FUNCTION_BLOCK FB 251
TITLE =G151M FRESH AIR LOUVER GERM 3
//COPYRIGHT:    (C) 2009  BUHLER AG, CH-9240 UZWIL, SWITZERLAND
//
//PRODUCT:      WinCoS_BIW01_09
//
//TITLE:        FRESH AIR LOUVER GERM 3
//                Machine group control
//                Maschinengruppensteuerung
//
//--------------------------------------------------------------------------------
//
//IDENT:        AUTHOR:             DEPT:                              DATE:
//
//P01_FB251.1.0 K.Renz              CSB41                              13.Jan.2010
//             1st Release
//
//--------------------------------------------------------------------------------
//
//PURPOSE:
//
//MANUAL :
//
//RESTRICTIONS:
//
//--------------------------------------------------------------------------------
AUTHOR : KR
FAMILY : USW
VERSION : 9.9


VAR
  Gr : FB 10;	//Standard interface to group
  InOutValue1 : DINT ;	//Data for user
  InOutValue2 : DINT ;	//Data for user
  OutWayConflict : BOOL ;	//Data for user
  OutSelectionOk : BOOL ;	//Data for user
  CmdNewValue : BOOL ;	//Data for user
  CmdNewJob : BOOL ;	//Data for user
  OutCodeOK : BOOL ;	//Data for user
  InEndOfJob : BOOL ;	//Data for user
  staWayOk : BOOL ;	//Data for user
  EdgeStartRelease : BOOL ;	//Data for user
  USW8 : BOOL ;	//Data for user
  USW9 : BOOL ;	//Data for user
  USW10 : BOOL ;	//Data for user
  USW11 : BOOL ;	//Data for user
  USW12 : BOOL ;	//Data for user
  USW13 : BOOL ;	//Data for user
  USW14 : BOOL ;	//Data for user
  USW15 : BOOL ;	//Data for user
  A_2351_BZS01 : FB 14;	// DigInpCont
  A_2351_BZS02 : FB 14;	// DigInpCont
  A_2351_MXZ01 : FB 20;	// VLS4Ctrl
  A_2352_BZS01 : FB 14;	// DigInpCont
  A_2352_BZS02 : FB 14;	// DigInpCont
  A_2352_MXZ01 : FB 20;	// VLS4Ctrl
END_VAR
VAR_TEMP
  tmpEnable : BOOL ;
  tmpFlag : BOOL ;
  tmpCmdNext : BOOL ;
  tmpLocal : BOOL ;
  tmpAspOk : BOOL ;
  tmpHWStop : BOOL ;
  tmpInstanzDBNo : INT ;
END_VAR
BEGIN
NETWORK
TITLE =



NETWORK
TITLE =Read command from group control
//Parameter
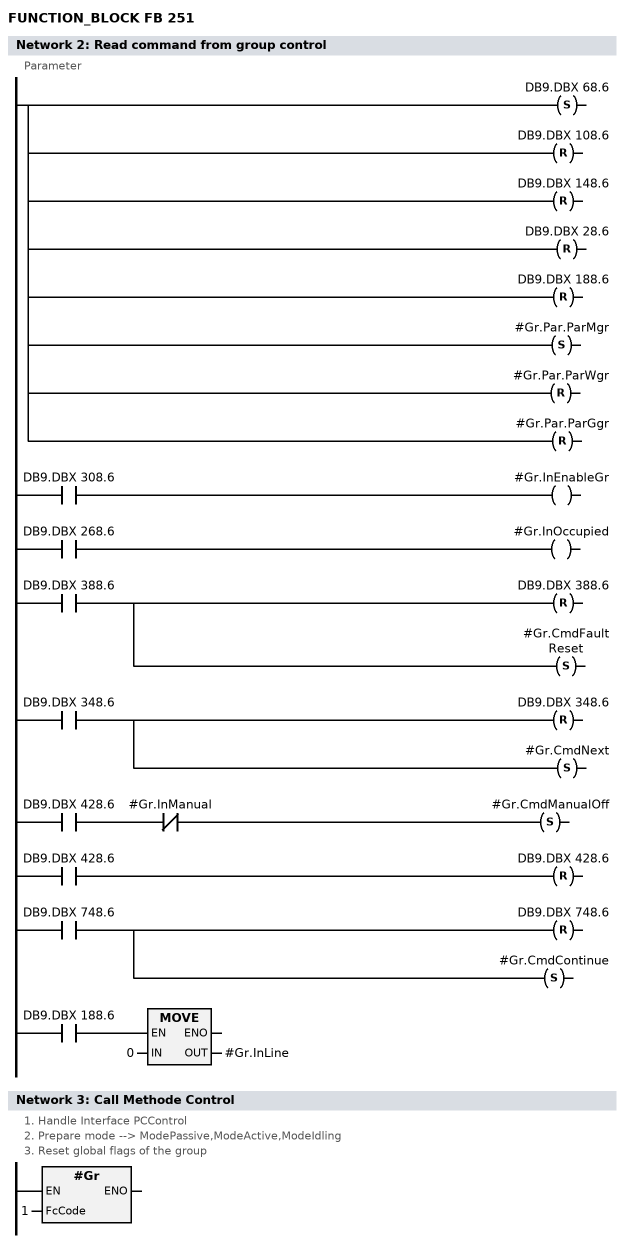
      SET   ;
      S     DB9.DBX   68.6;
      R     DB9.DBX  108.6;
      R     DB9.DBX  148.6;
      R     DB9.DBX   28.6;
      R     DB9.DBX  188.6;
      S     #Gr.Par.ParMgr;
      R     #Gr.Par.ParWgr;
      R     #Gr.Par.ParGgr;
//Command
      A     DB9.DBX  308.6;
      =     #Gr.InEnableGr;
      A     DB9.DBX  268.6;
      =     #Gr.InOccupied;
      A     DB9.DBX  388.6;
      R     DB9.DBX  388.6;
      S     #Gr.CmdFaultReset;
      A     DB9.DBX  348.6;
      R     DB9.DBX  348.6;
      S     #Gr.CmdNext;

      A     DB9.DBX  428.6;
      AN    #Gr.InManual;
      S     #Gr.CmdManualOff;
      A     DB9.DBX  428.6;
      R     DB9.DBX  428.6;

//      U     "GCS7_GrCtrlDB".CmdManualOff[151]
//      O     "GCS7_GrCtrlDB".OutOccupied[151]
//      R     "GCS7_GrCtrlDB".CmdManualOff[151]
//      S     #Gr.CmdManualOff

      A     DB9.DBX  748.6;
      R     DB9.DBX  748.6;
      S     #Gr.CmdContinue;
//Init Line Number
      A     DB9.DBX  188.6;
      JCN   WE00;
      L     0;
      T     #Gr.InLine;
WE00: NOP   0;
NETWORK
TITLE =Call Methode Control
// 1. Handle Interface PCControl
// 2. Prepare mode --> ModePassive,ModeActive,ModeIdling
// 3. Reset global flags of the group
      CALL #Gr (
           FcCode                   := 1);
NETWORK
TITLE =Restart Idling Time

      L     #Gr.Par.ParIdling;
      L     2;
      >=I   ;
      JC    IdTm;
      T     #Gr.Par.ParIdling;
IdTm: NOP   0;
      CLR   ;
      S     #Gr.CmdRestartIdling;
NETWORK
TITLE =Prepare global flags



NETWORK
TITLE =Set Pattern (Target position)

      A     #Gr.InManual;
      JC    ILO6;
      L     0; // 0.0%
      O     DB819.DBX  111.6;
      O     DB819.DBX  111.0;
      JC    PE;
      A     DB909.DBX  410.0;
      O(    ;
      A     DB909.DBX  412.1; // germinating Process finished
      AN    DB819.DBX  111.4;
      )     ;
      JCN   M003;
      NOP   0;
//BRT100310      L     "MAL1S019Par".StepAct.PosFreshAirFlapBasic
//      L     "MAL1S019Par".Par.ParIntMachine.TargetPosFreshAir    //BRT100310
//      L     10                          // convert to 0.1%
//      *I
PE:   NOP   0;

      A     DB251.DBX  131.5;
      JC    Man1;
      L     DB909.DBW  352; //BRT100310
      L     10; // convert to 0.1%
      *I    ;
      T     #A_2351_MXZ01.InPositionMiddle; // setpoint element
//-> 26.02.2014 IS. Start regulating from current position when switch to automatic
Man1: L     #A_2351_MXZ01.InPositionMiddle;
      L     10;
      /D    ;
      T     DB909.DBW  352;
//<-
      NOP   0;

      A     DB251.DBX  259.5;
      JC    Man2;
      L     DB909.DBW  254; // Target Position FreshAir 2
      L     10; // convert to 0.1%
      *I    ;
      T     #A_2352_MXZ01.InPositionMiddle; // setpoint element
//-> 26.02.2014 IS. Start regulating from current position when switch to automatic
Man2: L     #A_2352_MXZ01.InPositionMiddle;
      L     10;
      /D    ;
      T     DB909.DBW  254;
//<-
M003: NOP   0;
      JU    En06;
ILO6: NOP   0;
      L     DB909.DBW  230;
      L     10; // convert to 0.1%
      *I    ;
      T     #A_2351_MXZ01.InPositionMiddle; // setpoint element
      T     #A_2352_MXZ01.InPositionMiddle; // setpoint element
En06: NOP   0;



NETWORK
TITLE =Interlocking WayOk



NETWORK
TITLE =Interlocking Autostart

      CLR   ;
      R     #Gr.OutAutostart;
NETWORK
TITLE =Interlocking Enable
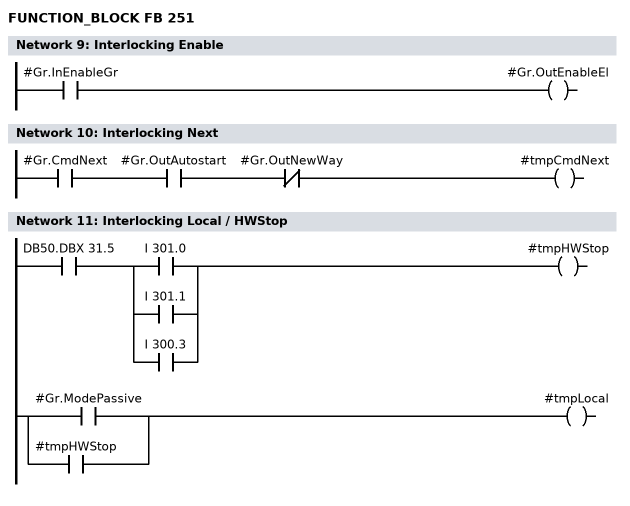

      A     #Gr.InEnableGr;
      =     #Gr.OutEnableEl;

NETWORK
TITLE =Interlocking Next

      A     #Gr.CmdNext;
      A     #Gr.OutAutostart;
      AN    #Gr.OutNewWay;
      =     #tmpCmdNext;

NETWORK
TITLE =Interlocking Local / HWStop

      A     DB50.DBX   31.5;
//BRT100310 - HW-Stop nur bei NOT-AUS +C23 oder Customer, nicht bei NOT-AUS Maschine!
      A(    ;
      O     I    301.0;
      O     I    301.1;
      O     I    300.3;
      )     ;
      =     #tmpHWStop;

      A     #Gr.ModePassive;
      O     #tmpHWStop;
      =     #tmpLocal;

NETWORK
TITLE ==A-2351-BZS01 : FRESH AIR FLAP 1 100% CIRCULATION AIR

      NOP   0;
//-InLocal---
      A     #tmpLocal;
      =     #A_2351_BZS01.InLocal;
//
//-Monitoring---
      CLR   ;
      =     #A_2351_BZS01.InMonTrue;
      CLR   ;
      =     #A_2351_BZS01.InMonFalse;
//
//-PreAlarm---
      CLR   ;
      =     #A_2351_BZS01.InPreAlarmTrue;
      CLR   ;
      =     #A_2351_BZS01.InPreAlarmFalse;
//
//-Additional commands---
//      CLR
//      S     #A_2351_BZS01.CmdRunTimeOutTime
//
//-Read inputs---
      A     I    364.6;
      =     #A_2351_BZS01.InpTrue;
      A     DB51.DBX    4.5;
      =     #A_2351_BZS01.InDPFault;
//
//-Set Parameters---
//
//-Call object control---
      CALL #A_2351_BZS01 ;
//
//-Write outputs---
NETWORK
TITLE ==A-2351-BZS02 : FRESH AIR FLAP 1 100% FRESH AIR

      NOP   0;
//-InLocal---
      A     #tmpLocal;
      =     #A_2351_BZS02.InLocal;
//
//-Monitoring---
      CLR   ;
      =     #A_2351_BZS02.InMonTrue;
      CLR   ;
      =     #A_2351_BZS02.InMonFalse;
//
//-PreAlarm---
      CLR   ;
      =     #A_2351_BZS02.InPreAlarmTrue;
      CLR   ;
      =     #A_2351_BZS02.InPreAlarmFalse;
//
//-Additional commands---
//      CLR
//      S     #A_2351_BZS02.CmdRunTimeOutTime
//
//-Read inputs---
      A     I    364.7;
      =     #A_2351_BZS02.InpTrue;
      A     DB51.DBX    4.5;
      =     #A_2351_BZS02.InDPFault;
//
//-Set Parameters---
//
//-Call object control---
      CALL #A_2351_BZS02 ;
//
//-Write outputs---
NETWORK
TITLE ==A-2351-MXZ01 : FRESH AIR FLAP 1

      NOP   0;
//-InLocal---
      A(    ;
      A     #tmpLocal;
      O     ;
      A     #Gr.InManual;
      AN    #Gr.InOutAutostartMan;
      )     ;
      A     #A_2351_MXZ01.StLN;
      =     #A_2351_MXZ01.InLocal;

//-Interlocking---
      A     #A_2351_MXZ01.Par.ParManual;
      A     #A_2351_MXZ01.InManual;
      JC    man1;
      A(    ;
      L     0;
      L     #A_2351_MXZ01.InPositionMiddle; // setpoint element
      ==I   ;
      )     ;
      A(    ;
      A     #Gr.InManual;
      A     #Gr.InOutAutostartMan;
      ON    #Gr.InManual;
      )     ;
      A     #Gr.OutEnableEl;
      =     #A_2351_MXZ01.InLN;

      A(    ;
      L     #A_2351_MXZ01.InPositionMiddle; // setpoint element
      L     0;
      >I    ;
      )     ;
      A(    ;
      L     #A_2351_MXZ01.InPositionMiddle; // setpoint element
      L     1000; // 100,0%
      <I    ;
      )     ;
      A(    ;
      A     #Gr.InManual;
      A     #Gr.InOutAutostartMan;
      ON    #Gr.InManual;
      )     ;
      A     #Gr.OutEnableEl;
      S     #A_2351_MXZ01.CmdMiddle1;

      CLR   ;
      =     #A_2351_MXZ01.CmdMiddle2;

      A(    ;
      AN    #Gr.InOccupied;
      AN    #Gr.InManual;
      )     ;
      O(    ;
      L     #A_2351_MXZ01.InPositionMiddle; // setpoint element
      L     1000; // 100,0%
      >=I   ;
      )     ;
      A(    ;
      A     #Gr.InManual;
      A     #Gr.InOutAutostartMan;
      ON    #Gr.InManual;
      )     ;
      A     #Gr.OutEnableEl;
      S     #A_2351_MXZ01.CmdHN;
man1: NOP   0;
//
//-Read inputs---
//====>BRT060310 - Regeln auf Zeit, ohne Auswertung Rückmeldung
      A     I    364.6;
      =     DB251.DBX  130.4;
      CLR   ;
      =     DB251.DBX  130.5;
      A     I    364.7;
      =     DB251.DBX  130.7;

//      U     #A_2351_BZS02.StTrue        // 100% Frischluft
//      SPBN  FL1
//      L     1000
//      SPA   INP1
//FL1:  NOP   0
//      U     #A_2351_BZS01.StTrue        // 100% Umluft
//      SPBN  RL1
//      L     0
//      SPA   INP1
//RL1:  NOP   0
//      L     "A_2351_BEE01_AI1"
//INP1: T     #A_2351_MXZ01.InpPosition
//<====BRT060310
//BRT110310      U     "PLC_SystemDB".HardwareStop.Germinating_3
      A     #tmpHWStop; //BRT110310
      =     #A_2351_MXZ01.InHWStop;
      A     DB51.DBX    4.5;
      =     #A_2351_MXZ01.InDPFault;
//
//-Set Parameters---
//
//-Call object control---
      CALL #A_2351_MXZ01 ;
//
//-Write outputs---
      A     #A_2351_MXZ01.OutpLN;
      =     Q    364.5;
      A     #A_2351_MXZ01.OutpHN;
      =     Q    364.4;

NETWORK
TITLE ==A-2352-BZS02 : FRESH AIR FLAP 2 100% FRESH AIR

      NOP   0;
//-InLocal---
      A     #tmpLocal;
      =     #A_2352_BZS02.InLocal;
//
//-Monitoring---
      CLR   ;
      =     #A_2352_BZS02.InMonTrue;
      CLR   ;
      =     #A_2352_BZS02.InMonFalse;
//
//-PreAlarm---
      CLR   ;
      =     #A_2352_BZS02.InPreAlarmTrue;
      CLR   ;
      =     #A_2352_BZS02.InPreAlarmFalse;
//
//-Additional commands---
//      CLR
//      S     #A_2352_BZS02.CmdRunTimeOutTime
//
//-Read inputs---
      A     I    365.3;
      =     #A_2352_BZS02.InpTrue;
      A     DB51.DBX    4.5;
      =     #A_2352_BZS02.InDPFault;
//
//-Set Parameters---
//
//-Call object control---
      CALL #A_2352_BZS02 ;
//
//-Write outputs---
NETWORK
TITLE ==A-2352-BZS01 : FRESH AIR FLAP 2 100% CIRCULATION AIR

      NOP   0;
//-InLocal---
      A     #tmpLocal;
      =     #A_2352_BZS01.InLocal;
//
//-Monitoring---
      CLR   ;
      =     #A_2352_BZS01.InMonTrue;
      CLR   ;
      =     #A_2352_BZS01.InMonFalse;
//
//-PreAlarm---
      CLR   ;
      =     #A_2352_BZS01.InPreAlarmTrue;
      CLR   ;
      =     #A_2352_BZS01.InPreAlarmFalse;
//
//-Additional commands---
//      CLR
//      S     #A_2352_BZS01.CmdRunTimeOutTime
//
//-Read inputs---
      A     I    365.2;
      =     #A_2352_BZS01.InpTrue;
      A     DB51.DBX    4.5;
      =     #A_2352_BZS01.InDPFault;
//
//-Set Parameters---
//
//-Call object control---
      CALL #A_2352_BZS01 ;
//
//-Write outputs---
NETWORK
TITLE ==A-2352-MXZ01 : FRESH AIR FLAP 2

      NOP   0;
//-InLocal---
      A(    ;
      A     #tmpLocal;
      O     ;
      A     #Gr.InManual;
      AN    #Gr.InOutAutostartMan;
      )     ;
      A     #A_2352_MXZ01.StLN;
      =     #A_2352_MXZ01.InLocal;

//-Interlocking---
      A     #A_2352_MXZ01.Par.ParManual;
      A     #A_2352_MXZ01.InManual;
      JC    man2;
      A(    ;
      L     0;
      L     #A_2352_MXZ01.InPositionMiddle; // setpoint element
      ==I   ;
      )     ;
      A(    ;
      A     #Gr.InManual;
      A     #Gr.InOutAutostartMan;
      ON    #Gr.InManual;
      )     ;
      A     #Gr.OutEnableEl;
      =     #A_2352_MXZ01.InLN;

      A(    ;
      L     #A_2352_MXZ01.InPositionMiddle; // setpoint element
      L     0;
      >I    ;
      )     ;
      A(    ;
      L     #A_2352_MXZ01.InPositionMiddle; // setpoint element
      L     1000; // 100,0%
      <I    ;
      )     ;
      A(    ;
      A     #Gr.InManual;
      A     #Gr.InOutAutostartMan;
      ON    #Gr.InManual;
      )     ;
      A     #Gr.OutEnableEl;
      S     #A_2352_MXZ01.CmdMiddle1;

      CLR   ;
      =     #A_2352_MXZ01.CmdMiddle2;

      A(    ;
      AN    #Gr.InOccupied;
      AN    #Gr.InManual;
      )     ;
      O(    ;
      L     #A_2352_MXZ01.InPositionMiddle; // setpoint element
      L     1000; // 100,0%
      >=I   ;
      )     ;
      A(    ;
      A     #Gr.InManual;
      A     #Gr.InOutAutostartMan;
      ON    #Gr.InManual;
      )     ;
      A     #Gr.OutEnableEl;
      S     #A_2352_MXZ01.CmdHN;
man2: NOP   0;
//
//-Read inputs---
//====>BRT060310 - Regeln auf Zeit, ohne Auswertung Rückmeldung
      A     I    365.2;
      =     DB251.DBX  258.4;
      CLR   ;
      =     DB251.DBX  258.5;
      A     I    365.3;
      =     DB251.DBX  258.7;

//      U     #A_2352_BZS02.StTrue        // 100% Frischluft
//      SPBN  FL2
//      L     1000
//      SPA   INP2
//FL2:  NOP   0
//      U     #A_2352_BZS01.StTrue        // 100% Umluft
//      SPBN  RL2
//      L     0
//      SPA   INP2
//RL2:  NOP   0
//      L     "A_2352_BEE01_AI1"
//INP2: T     #A_2352_MXZ01.InpPosition
//<====BRT100310
//BRT110310      U     "PLC_SystemDB".HardwareStop.Germinating_3
      A     #tmpHWStop; //BRT110310
      =     #A_2352_MXZ01.InHWStop;
      A     DB51.DBX    4.5;
      =     #A_2352_MXZ01.InDPFault;
//
//-Set Parameters---
//
//-Call object control---
      CALL #A_2352_MXZ01 ;
//
//-Write outputs---
      A     #A_2352_MXZ01.OutpLN;
      =     Q    365.1;
      A     #A_2352_MXZ01.OutpHN;
      =     Q    365.0;

NETWORK
TITLE =Test Fault
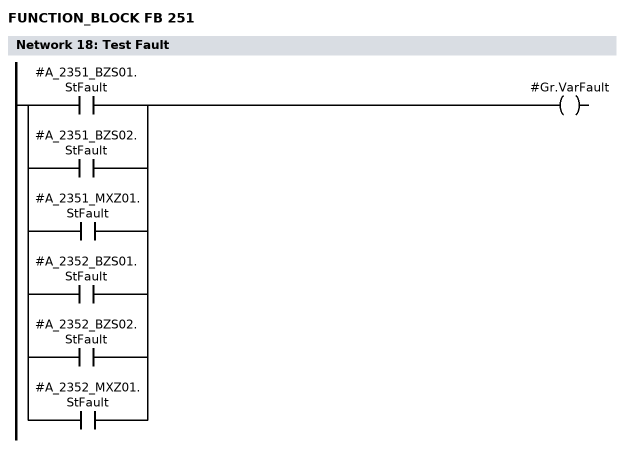

      A     #A_2351_BZS01.StFault;
      O     #A_2351_BZS02.StFault;
      O     #A_2351_MXZ01.StFault;
      O     #A_2352_BZS01.StFault;
      O     #A_2352_BZS02.StFault;
      O     #A_2352_MXZ01.StFault;
      =     #Gr.VarFault;
NETWORK
TITLE =Test Warning

      CLR   ;
      =     #Gr.OutWarning;
NETWORK
TITLE =Test Stopped
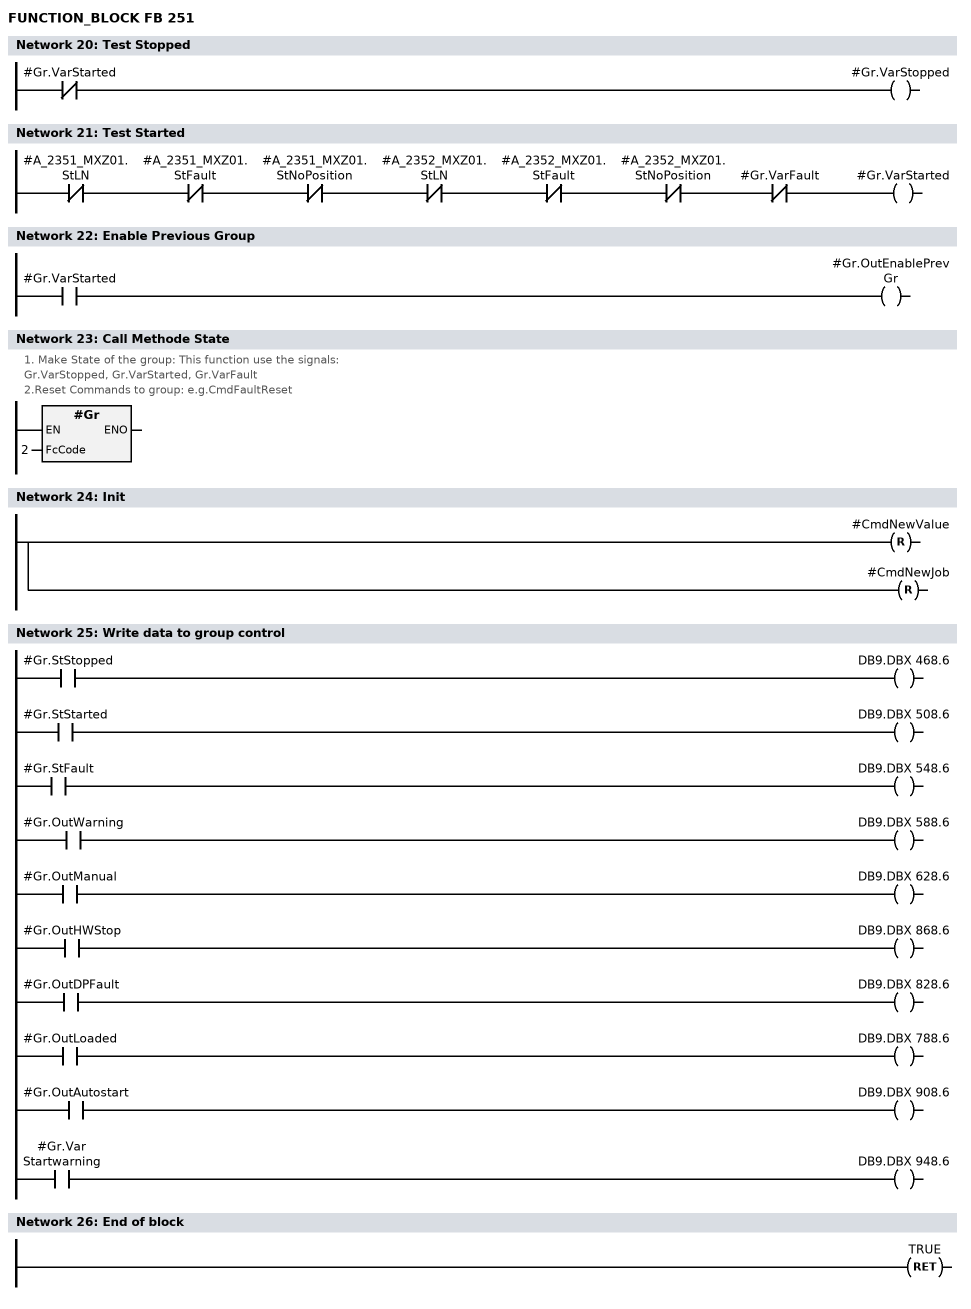

//BRT100310       U     #A_2351_MXZ01.StLN
//BRT100310       U     #A_2352_MXZ01.StLN
//BRT100310       UN    #Gr.VarFault
      AN    #Gr.VarStarted;
      =     #Gr.VarStopped;
NETWORK
TITLE =Test Started

      AN    #A_2351_MXZ01.StLN;
      AN    #A_2351_MXZ01.StFault;
      AN    #A_2351_MXZ01.StNoPosition;
      AN    #A_2352_MXZ01.StLN;
      AN    #A_2352_MXZ01.StFault;
      AN    #A_2352_MXZ01.StNoPosition;
//BRT100310      UN    #Gr.VarStopped
      AN    #Gr.VarFault;
      =     #Gr.VarStarted;
NETWORK
TITLE =Enable Previous Group

      A     #Gr.VarStarted;
      =     #Gr.OutEnablePrevGr;
NETWORK
TITLE =Call Methode State
//1. Make State of the group: This function use the signals:
//        Gr.VarStopped, Gr.VarStarted, Gr.VarFault
//2.Reset Commands to group: e.g.CmdFaultReset
      CALL #Gr (
           FcCode                   := 2);
NETWORK
TITLE =Init

      SET   ;
      R     #CmdNewValue;
      R     #CmdNewJob;
NETWORK
TITLE =Write data to group control

      A     #Gr.StStopped;
      =     DB9.DBX  468.6;
      A     #Gr.StStarted;
      =     DB9.DBX  508.6;
      A     #Gr.StFault;
      =     DB9.DBX  548.6;
      A     #Gr.OutWarning;
      =     DB9.DBX  588.6;
      A     #Gr.OutManual;
      =     DB9.DBX  628.6;
      A     #Gr.OutHWStop;
      =     DB9.DBX  868.6;
      A     #Gr.OutDPFault;
      =     DB9.DBX  828.6;
      A     #Gr.OutLoaded;
      =     DB9.DBX  788.6;
      A     #Gr.OutAutostart;
      =     DB9.DBX  908.6;
      A     #Gr.VarStartwarning;
      =     DB9.DBX  948.6;
NETWORK
TITLE =End of block

      BE    ;

END_FUNCTION_BLOCK

